INTERFACE I_OutputPorts

METHOD PUBLIC Accept
VAR_INPUT
	Visitor : I_OutputPortVisitor;
END_VAR
END_METHOD

METHOD PUBLIC AddDataAsOutputPort : I_OutputPort
VAR_INPUT
	Name : T_MAXSTRING;
	Data : I_Datatype;
END_VAR
END_METHOD

METHOD AddOutputPort
VAR_INPUT
	OutputPort : I_OutputPort;
END_VAR
END_METHOD

PROPERTY PUBLIC HasOutputPorts : BOOL
GET
END_GET
END_PROPERTY

METHOD PUBLIC TryGetOutputPortByName : BOOL
VAR_INPUT
	Name : T_MAXSTRING;
	Destination : REFERENCE TO I_OutputPort;
END_VAR
END_METHOD

END_INTERFACE

(* stored: Version 1.1.0.1, ProductVersion 3.1.4024.12
   Itf I_OutputPorts: Id {7106d115-8795-4b25-8759-763d1e526662}
   Method Accept: Id {79fdd00f-4f69-4c1b-a985-c60d009ac80a}
   Method AddDataAsOutputPort: Id {123eab4b-32fd-4da5-9fe0-541c899fba27}
   Method AddOutputPort: Id {9cf945e5-debb-4ba1-b08e-ce2d568d025a}
   Property HasOutputPorts: Id {6054b98a-c133-025c-1121-f3967a211dc4}
   Get Get: Id {5c0b444f-288b-0201-25cb-f63026639d21}
   Method TryGetOutputPortByName: Id {a51707f2-05d5-44f8-bd48-066fefa88e9c} *)
